Staubli VAL3: cleanUserMenu.pgx

program cleanUserMenu()
  local num i
begin
//  // clean all the reference
//  for i=0 to size(sMenuUser)-1
//    sMenuUser[i]=""
//  endFor
end
